FUNCTION F_RealIsValid : BOOL
VAR_INPUT
	rInput			: REAL;
END_VAR
VAR
	refReal			: REFERENCE TO REAL;
END_VAR

refReal		REF= rInput;

IF RealIsNan(refReal) THEN
	F_RealIsValid	:= FALSE;
	RETURN;
ELSE
	IF (ABS(refReal) < EXP(-10) AND refReal <> 0) OR ABS(refReal) > EXP(10) THEN
		F_RealIsValid	:= FALSE;
		RETURN;
	ELSE
		F_RealIsValid	:= TRUE;
		RETURN;
	END_IF
END_IF

END_FUNCTION

(* stored: Version 1.1.0.1, ProductVersion 3.1.4024.12
   POU F_RealIsValid: Id {46b2d020-203a-40ee-9103-5ad37c363a44}, SpecialFunc None *)
